FUNCTION_BLOCK PEView (* Composite Function Block Type *)
  (* Standard: 61499-2 *)
  (* Version 0.2, 2003-12-05, JHC, Rockwell Automation, Renamed from NEWCOMPFB. *)
  (* Version 0.1, 2002-01-08, JHC, Rockwell Automation, Added DLY FB as example. *)
  (* Version 0.0, 2000-05-27, JHC, Rockwell Automation *)
  (* Compiler header: package fb.rt.cs725;import fb.rt.vhmi.*; *)
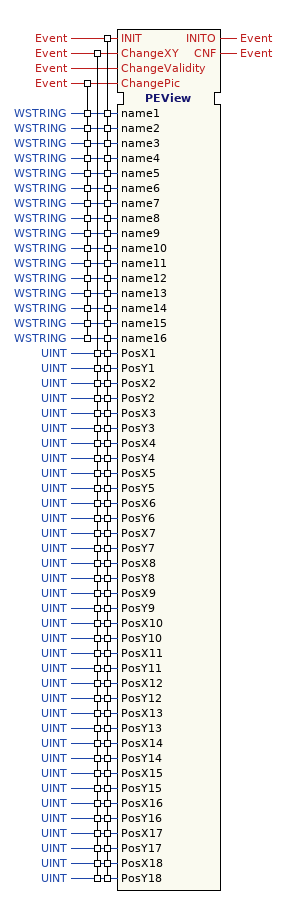
  EVENT_INPUT
    INIT WITH PosX1, PosY1, PosX2, PosY2, PosX3, PosY3, PosX4, PosY4, PosX5, PosY5, PosX6, PosY6, PosX7, PosY7, PosX8, PosY8, PosX9, PosY9, PosX10, PosY10, PosX11, PosY11, PosX12, PosY12, PosX13, PosY13, PosX14, PosY14, PosX15, PosY15, PosX16, PosY16, PosX17, PosY17, PosX18, PosY18, name1, name2, name3, name4, name5, name6, name7, name8, name9, name10, name11, name12, name13, name14, name15, name16; (* Initialization Request *)
    ChangeXY WITH PosX1, PosY1, PosX2, PosY2, PosX3, PosY3, PosX4, PosY4, PosX5, PosY5, PosX6, PosY6, PosX7, PosY7, PosX8, PosY8, PosX9, PosY9, PosX10, PosY10, PosX11, PosY11, PosX12, PosY12, PosX13, PosY13, PosX14, PosY14, PosX15, PosY15, PosX16, PosY16, PosX17, PosY17, PosX18, PosY18; (* Normal Execution Request *)
    ChangeValidity;
    ChangePic WITH name1, name2, name3, name4, name5, name6, name7, name8, name9, name10, name11, name12, name13, name14, name15, name16;
  END_EVENT
  EVENT_OUTPUT
    INITO; (* Initialization Confirm *)
    CNF; (* Execution Confirmation *)
  END_EVENT
  VAR_INPUT
    name1 : WSTRING;
    name2 : WSTRING;
    name3 : WSTRING;
    name4 : WSTRING;
    name5 : WSTRING;
    name6 : WSTRING;
    name7 : WSTRING;
    name8 : WSTRING;
    name9 : WSTRING;
    name10 : WSTRING;
    name11 : WSTRING;
    name12 : WSTRING;
    name13 : WSTRING;
    name14 : WSTRING;
    name15 : WSTRING;
    name16 : WSTRING;
    PosX1 : UINT;
    PosY1 : UINT;
    PosX2 : UINT;
    PosY2 : UINT;
    PosX3 : UINT;
    PosY3 : UINT;
    PosX4 : UINT;
    PosY4 : UINT;
    PosX5 : UINT;
    PosY5 : UINT;
    PosX6 : UINT;
    PosY6 : UINT;
    PosX7 : UINT;
    PosY7 : UINT;
    PosX8 : UINT;
    PosY8 : UINT;
    PosX9 : UINT;
    PosY9 : UINT;
    PosX10 : UINT;
    PosY10 : UINT;
    PosX11 : UINT;
    PosY11 : UINT;
    PosX12 : UINT;
    PosY12 : UINT;
    PosX13 : UINT;
    PosY13 : UINT;
    PosX14 : UINT;
    PosY14 : UINT;
    PosX15 : UINT;
    PosY15 : UINT;
    PosX16 : UINT;
    PosY16 : UINT;
    PosX17 : UINT;
    PosY17 : UINT;
    PosX18 : UINT;
    PosY18 : UINT;
  END_VAR
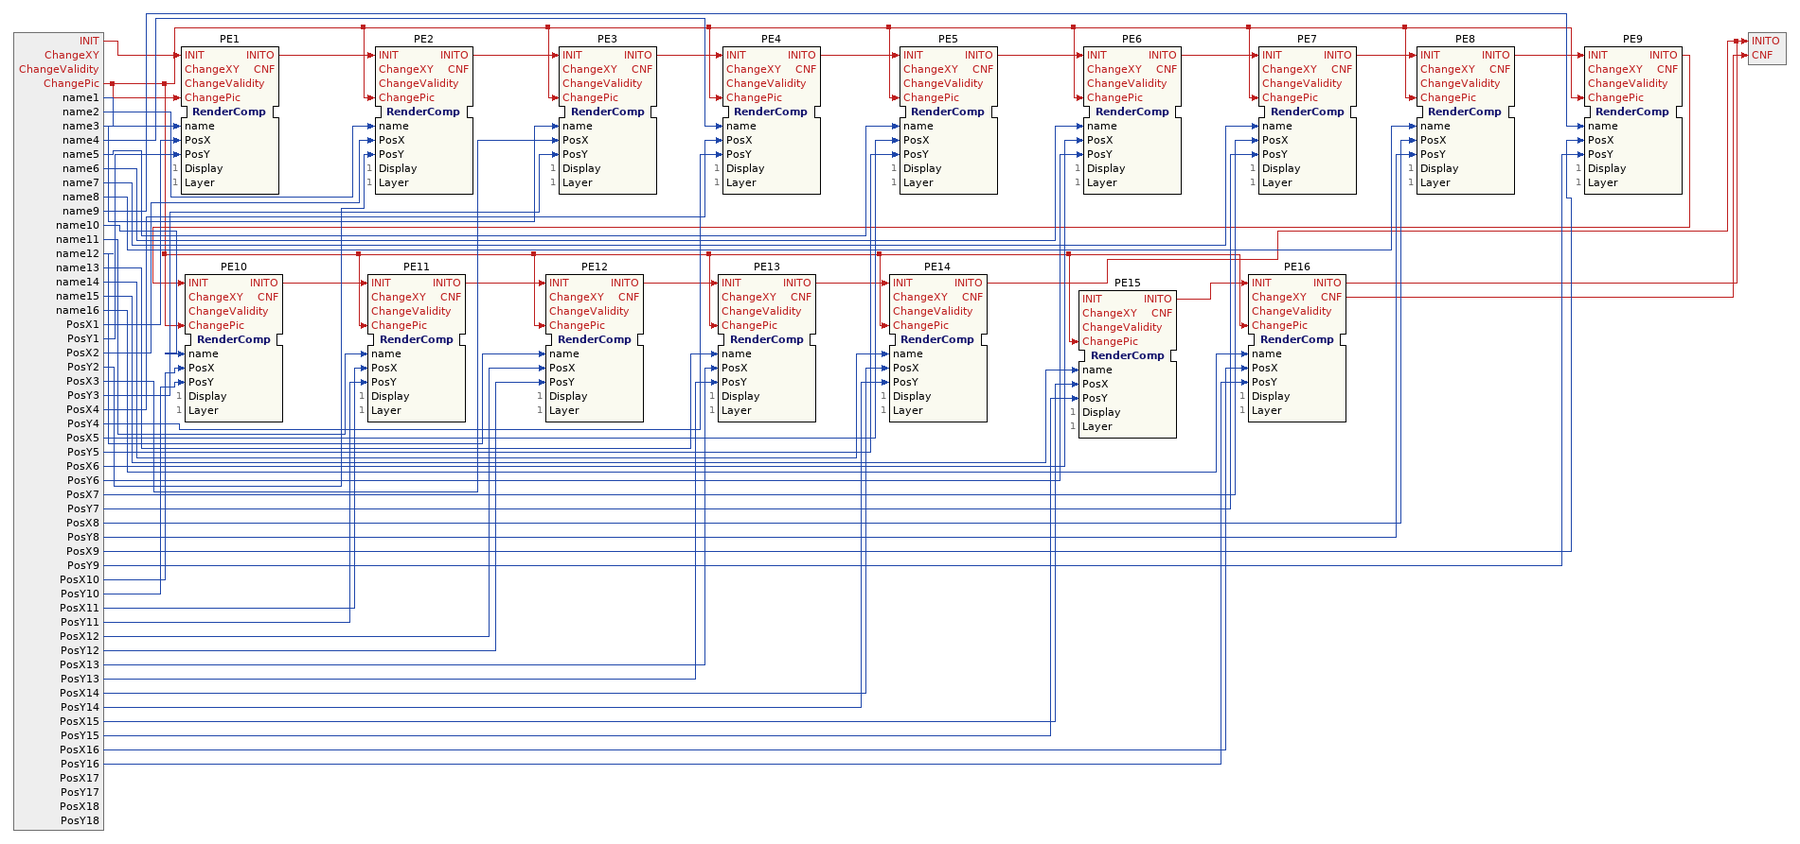
  FBS
    PE1 : RenderComp(Layer := 1, Display := 1);
    PE2 : RenderComp(Layer := 1, Display := 1);
    PE3 : RenderComp(Layer := 1, Display := 1);
    PE4 : RenderComp(Layer := 1, Display := 1);
    PE5 : RenderComp(Layer := 1, Display := 1);
    PE6 : RenderComp(Layer := 1, Display := 1);
    PE7 : RenderComp(Layer := 1, Display := 1);
    PE8 : RenderComp(Layer := 1, Display := 1);
    PE9 : RenderComp(Layer := 1, Display := 1);
    PE10 : RenderComp(Layer := 1, Display := 1);
    PE11 : RenderComp(Layer := 1, Display := 1);
    PE12 : RenderComp(Layer := 1, Display := 1);
    PE13 : RenderComp(Layer := 1, Display := 1);
    PE14 : RenderComp(Layer := 1, Display := 1);
    PE15 : RenderComp(Layer := 1, Display := 1);
    PE16 : RenderComp(Layer := 1, Display := 1);
  END_FBS
  EVENT_CONNECTIONS
    INIT TO PE1.INIT;
    PE1.INITO TO PE2.INIT;
    PE2.INITO TO PE3.INIT;
    PE3.INITO TO PE4.INIT;
    PE4.INITO TO PE5.INIT;
    PE5.INITO TO PE6.INIT;
    PE6.INITO TO PE7.INIT;
    PE7.INITO TO PE8.INIT;
    PE8.INITO TO PE9.INIT;
    PE9.INITO TO PE10.INIT;
    PE10.INITO TO PE11.INIT;
    PE11.INITO TO PE12.INIT;
    PE12.INITO TO PE13.INIT;
    PE13.INITO TO PE14.INIT;
    PE15.INITO TO PE16.INIT;
    PE16.INITO TO INITO;
    PE16.CNF TO CNF;
    ChangePic TO PE1.ChangePic;
    ChangePic TO PE2.ChangePic;
    ChangePic TO PE3.ChangePic;
    ChangePic TO PE4.ChangePic;
    ChangePic TO PE5.ChangePic;
    ChangePic TO PE6.ChangePic;
    ChangePic TO PE7.ChangePic;
    ChangePic TO PE8.ChangePic;
    ChangePic TO PE9.ChangePic;
    ChangePic TO PE10.ChangePic;
    ChangePic TO PE11.ChangePic;
    ChangePic TO PE12.ChangePic;
    ChangePic TO PE13.ChangePic;
    ChangePic TO PE14.ChangePic;
    ChangePic TO PE15.ChangePic;
    ChangePic TO PE16.ChangePic;
    PE14.INITO TO INITO;
  END_CONNECTIONS
  DATA_CONNECTIONS
    PosX1 TO PE1.PosX;
    PosY1 TO PE1.PosY;
    PosX2 TO PE2.PosX;
    PosY2 TO PE2.PosY;
    PosX3 TO PE3.PosX;
    PosY3 TO PE3.PosY;
    PosX4 TO PE4.PosX;
    PosY4 TO PE4.PosY;
    PosX5 TO PE5.PosX;
    PosY5 TO PE5.PosY;
    PosX6 TO PE6.PosX;
    PosY6 TO PE6.PosY;
    PosX7 TO PE7.PosX;
    PosY7 TO PE7.PosY;
    PosX8 TO PE8.PosX;
    PosY8 TO PE8.PosY;
    PosX9 TO PE9.PosX;
    PosY9 TO PE9.PosY;
    PosX10 TO PE10.PosX;
    PosY10 TO PE10.PosY;
    PosX11 TO PE11.PosX;
    PosY11 TO PE11.PosY;
    PosX12 TO PE12.PosX;
    PosY12 TO PE12.PosY;
    PosX13 TO PE13.PosX;
    PosY13 TO PE13.PosY;
    PosX14 TO PE14.PosX;
    PosY14 TO PE14.PosY;
    PosX15 TO PE15.PosX;
    PosY15 TO PE15.PosY;
    PosX16 TO PE16.PosX;
    PosY16 TO PE16.PosY;
    name1 TO PE1.name;
    name2 TO PE2.name;
    name3 TO PE3.name;
    name4 TO PE4.name;
    name5 TO PE5.name;
    name6 TO PE6.name;
    name7 TO PE7.name;
    name8 TO PE8.name;
    name9 TO PE9.name;
    name10 TO PE10.name;
    name11 TO PE11.name;
    name12 TO PE12.name;
    name13 TO PE13.name;
    name14 TO PE14.name;
    name15 TO PE15.name;
    name16 TO PE16.name;
  END_CONNECTIONS
END_FUNCTION_BLOCK
